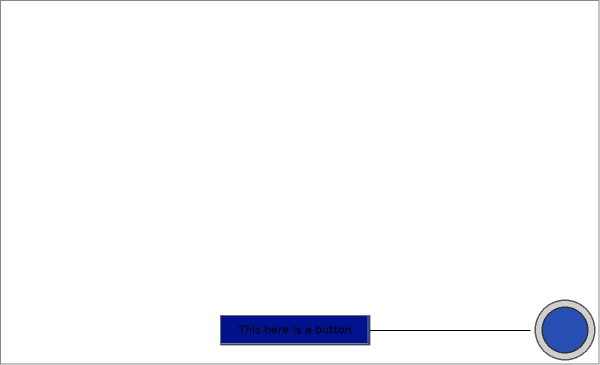
VISUALIZATION Visualization  // 600x365
    Button (220,315 150x30), "This here is a button", tooltip "Push to light the lamp"
        OnMouseDown: toggle MAIN._ButtonIsPushed
        OnMouseUp: toggle MAIN._ButtonIsPushed
    Lamp1 (530,295 70x70), variable: MAIN._LampIsOn, style: Lamp-Lamp1-Blue
    Line (370,330) (530,330)
END_VISUALIZATION

(* stored: Version 1.1.0.1
   Visu Visualization: Id {b34e380b-7928-4561-b0b3-e0bf8fa0b57f} *)
